FUNCTION_BLOCK FB_TransportBand
VAR_INPUT
	bEnable : BOOL;
	bExecute : BOOL;
	bHalt : BOOL;
END_VAR

VAR_OUTPUT
	eState : eBetriebszustand;
END_VAR
VAR
	nState : INT := 0;
	rVelocity : REAL;
	rAcceleration : REAL;
	bHaltStart : BOOL := FALSE; // Hilfsvariable, um Halt-Vorgang zu steuern
	// Motionblöcke der Tc2_Mc2
	mcReset : MC_Reset;
	mcPower : MC_Power;
	mcVelocity : MC_MoveVelocity;
	mcHalt : MC_Halt;
END_VAR

VAR_IN_OUT
	ax : Axis_Ref;
END_VAR

ax.ReadStatus();
mcReset(
	Axis:= ax, 
	Execute:= , 
	Done=> , 
	Busy=> , 
	Error=> , 
	ErrorID=> );
	
mcPower(
	Axis:= ax, 
	Enable:= , 
	Enable_Positive:= , 
	Enable_Negative:= , 
	Override:= , 
	BufferMode:= , 
	Options:= , 
	Status=> , 
	Busy=> , 
	Error=> , 
	ErrorID=> );

mcVelocity(
	Axis:= ax, 
	Execute:= , 
	Velocity:= 30, 
	Acceleration:= 60, 
	Deceleration:= , 
	Jerk:= , 
	Direction:= MC_Positive_Direction, 
	BufferMode:= , 
	Options:= , 
	InVelocity=> , 
	Busy=> , 
	Active=> , 
	CommandAborted=> , 
	Error=> , 
	ErrorID=> );
	
mcHalt(
	Axis:= ax, 
	Execute:= , 
	Deceleration:= 10, 
	Jerk:= , 
	BufferMode:= , 
	Options:= , 
	Done=> , 
	Busy=> , 
	Active=> , 
	CommandAborted=> , 
	Error=> , 
	ErrorID=> );

	

IF NOT mcPower.Status THEN
	nState := 0;
END_IF

CASE nState OF
	0: //OFF
	eState := eBetriebszustand.Off;
	mcPower.Enable := TRUE;
	mcPower.Enable_Positive := TRUE;
	//Fehler in der Init Logik
	IF bEnable AND mcPower.Status THEN
		nState := 20; //Ready
	ELSIF bEnable AND NOT mcPower.Status THEN
		nState := 10; // Init-Rest
	END_IF
	
	10: //Init - Reset
	eState := eBetriebszustand.Init;
	mcReset.Execute := TRUE;
	mcPower.Enable := FALSE;
	IF mcReset.Done THEN
		mcReset.Execute := FALSE;
		nState := 11;
	END_IF
	
	11: // Init - Power
	eState := eBetriebszustand.Init;
	mcPower.Enable := TRUE;
	mcReset.Execute := FALSE;
	IF mcPower.Status THEN
		nState := 20;
	END_IF
	
	20: //Ready
	eState := eBetriebszustand.Ready;
	IF bExecute THEN
		nState := 30;
	END_IF
	
	30: //Production
	eState := eBetriebszustand.Production;
	mcVelocity.Execute := TRUE;
	mcVelocity.Velocity := rVelocity;
	mcVelocity.Acceleration := rAcceleration;
	mcVelocity.Direction := MC_Positive_Direction;
	
	IF bHalt THEN 
		mcVelocity.Execute := FALSE;
		nState := 31;
	END_IF
	
	31: // Halten
	eState := eBetriebszustand.Production;
	//mcVelocity.Execute := FALSE;
	mcHalt.Execute := TRUE;
	mcHalt.CommandAborted;
	mcHalt.Active;
	mcHalt.Busy;
	mcHalt.Error;
	//mcVelocity.Acceleration := rAcceleration;
	IF mcHalt.Done THEN
		nState := 40;
	END_IF
	
	
	40: // Fertig
	eState := eBetriebszustand.Done;
	mcHalt.Execute := FALSE;
	//mcHalt.Deceleration := rAcceleration;
	
	IF NOT bExecute THEN
		nState := 20; 
	END_IF
END_CASE

END_FUNCTION_BLOCK

(* stored: Version 1.1.0.1, ProductVersion 3.1.4024.15
   POU FB_TransportBand: Id {2819a62a-8874-4d2c-b723-f866df5fb0bc}, SpecialFunc None *)
